(* IEC 61131-3 sources: Caravan/Stations/MachineControl/MachineControl/Class/TempControl_Class, 2 files *)

(* ---- TempControl_Class-TAB-EPM-01.st ---- *)
(*!
<Class
	Name               = "TempControl_Class"
	Revision           = "0.0"
	RealtimeTask       = "false"
	CyclicTask         = "true"
	BackgroundTask     = "false"
	Sigmatek           = "false"
	OSInterface        = "false"
	HighPriority       = "false"
	Automatic          = "false"
	UpdateMode         = "Prescan"
	SharedCommandTable = "true"
	Objectsize         = "(960,300)">
	<Channels>
		<Server Name="Actual_TempHZS_S" Visualized="true" Initialize="false" WriteProtected="false" Retentive="false"/>
		<Server Name="Actual_UltraheatTemp_S" Visualized="true" Initialize="false" WriteProtected="false" Retentive="false"/>
		<Server Name="ActualRoomTemp_S" Visualized="true" Initialize="false" WriteProtected="false" Retentive="false"/>
		<Server Name="ClassSvr" Visualized="false" Initialize="false" WriteProtected="true" Retentive="false"/>
		<Server Name="FanSpeed_S" Visualized="true" Initialize="true" DefValue="5" WriteProtected="false" Retentive="File"/>
		<Server Name="HeaterOn_S" Visualized="true" Initialize="false" WriteProtected="false" Retentive="File"/>
		<Server Name="SetRoomTemp_S" Visualized="true" Initialize="false" WriteProtected="false" Retentive="File"/>
		<Server Name="SetTempHZS_s" Visualized="true" Initialize="true" DefValue="200" WriteProtected="false" Retentive="File"/>
		<Client Name="ActualRoomTemp_C" Required="true" Internal="false"/>
		<Client Name="ActualUltraheatTemp_C" Required="true" Internal="false"/>
		<Client Name="HeaterRun_C" Required="true" Internal="false"/>
		<Client Name="MotorRunStop_C" Required="true" Internal="false"/>
		<Client Name="SetFanSpeed_C" Required="true" Internal="false"/>
		<Client Name="TempHZS_C" Required="true" Internal="false"/>
	</Channels>
</Class>
*)
TempControl_Class : CLASS
  //Servers:
	ClassSvr 	: SvrChCmd_DINT;
	Actual_TempHZS_S 	: SvrCh_DINT;
	ActualRoomTemp_S 	: SvrCh_DINT;
	Actual_UltraheatTemp_S 	: SvrCh_DINT;
	SetTempHZS_s 	: SvrCh_DINT;
	FanSpeed_S 	: SvrCh_DINT;
	SetRoomTemp_S 	: SvrCh_DINT;
	HeaterOn_S 	: SvrCh_DINT;
  //Clients:
	TempHZS_C 	: CltCh_DINT;
	ActualRoomTemp_C 	: CltCh_DINT;
	ActualUltraheatTemp_C 	: CltCh_DINT;
	SetFanSpeed_C 	: CltCh_DINT;
	MotorRunStop_C 	: CltCh_DINT;
	HeaterRun_C 	: CltCh_DINT;
  //Variables:
  //Functions:

	FUNCTION VIRTUAL GLOBAL CyWork
		VAR_INPUT
			EAX 	: UDINT;
		END_VAR
		VAR_OUTPUT
			state (EAX) 	: UDINT;
		END_VAR;
  //Tables:
	FUNCTION @STD
		VAR_OUTPUT
			ret_code	: CONFSTATES;
		END_VAR;
	FUNCTION GLOBAL TAB @CT_;
END_CLASS;

FUNCTION VIRTUAL GLOBAL TempControl_Class::CyWork
	VAR_INPUT
		EAX 	: UDINT;
	END_VAR
	VAR_OUTPUT
		state (EAX) 	: UDINT;
	END_VAR

    //Variablen einlesen
    TempHZS_C   :=    TempHZS_C.Read();

    ActualRoomTemp_C  :=  ActualRoomTemp_C.Read();

    ActualUltraheatTemp_C :=  ActualUltraheatTemp_C.Read();

    SetFanSpeed_C :=  SetFanSpeed_C.Read();

    MotorRunStop_C  :=  MotorRunStop_C.Read();

    HeaterRun_C :=  HeaterRun_C.Read();

    //Temperatur steuern
    if ActualRoomTemp_C < (SetRoomTemp_S - 1) & HeaterOn_S  = 1 then

        HeaterRun_C :=  1;

      elsif ActualRoomTemp_C > SetRoomTemp_S | HeaterOn_S = 0 then

        HeaterRun_C :=  0;

    end_if;

     //Variablen Schreiben
     Actual_TempHZS_S   :=    Actual_TempHZS_S.Write(input:=TempHZS_C);
     ActualRoomTemp_S   :=    ActualRoomTemp_S.Write(input:=ActualRoomTemp_C);

	state := READY;

END_FUNCTION

(* ---- TempControl_Class.st ---- *)
(*!
<Class
	Name               = "TempControl_Class"
	Revision           = "0.0"
	RealtimeTask       = "false"
	CyclicTask         = "true"
	BackgroundTask     = "false"
	Sigmatek           = "false"
	OSInterface        = "false"
	HighPriority       = "false"
	Automatic          = "false"
	UpdateMode         = "Prescan"
	SharedCommandTable = "true"
	Objectsize         = "(960,300)">
	<Channels>
		<Server Name="Actual_TempHZS_S" Visualized="true" Initialize="false" WriteProtected="false" Retentive="false"/>
		<Server Name="Actual_UltraheatTemp_S" Visualized="true" Initialize="false" WriteProtected="false" Retentive="false"/>
		<Server Name="ActualRoomTemp_S" Visualized="true" Initialize="false" WriteProtected="false" Retentive="false"/>
		<Server Name="ClassSvr" Visualized="false" Initialize="false" WriteProtected="true" Retentive="false"/>
		<Server Name="FanMode_S" Visualized="true" Initialize="false" WriteProtected="false" Retentive="File"/>
		<Server Name="FanSpeed_S" Visualized="true" Initialize="true" DefValue="5" WriteProtected="false" Retentive="File"/>
		<Server Name="HeaterOn_S" Visualized="true" Initialize="false" WriteProtected="false" Retentive="File"/>
		<Server Name="SetRoomTemp_S" Visualized="true" Initialize="false" WriteProtected="false" Retentive="File"/>
		<Server Name="SetTempHZS_s" Visualized="true" Initialize="true" DefValue="200" WriteProtected="false" Retentive="File"/>
		<Client Name="ActualRoomTemp_C" Required="true" Internal="false"/>
		<Client Name="ActualUltraheatTemp_C" Required="true" Internal="false"/>
		<Client Name="Heater200Watt_C" Required="true" Internal="false"/>
		<Client Name="HeaterOn_C" Required="true" Internal="false" DefValue="0"/>
		<Client Name="HeaterRun_C" Required="true" Internal="false" DefValue="0"/>
		<Client Name="MotorRunStop_C" Required="true" Internal="false"/>
		<Client Name="SetFanSpeed_C" Required="true" Internal="false"/>
		<Client Name="TempHZS_C" Required="true" Internal="false"/>
	</Channels>
</Class>
*)
TempControl_Class : CLASS
  //Servers:
	ClassSvr 	: SvrChCmd_DINT;
	Actual_TempHZS_S 	: SvrCh_DINT;
	ActualRoomTemp_S 	: SvrCh_DINT;
	Actual_UltraheatTemp_S 	: SvrCh_DINT;
	SetTempHZS_s 	: SvrCh_DINT;
	SetRoomTemp_S 	: SvrCh_DINT;
	HeaterOn_S 	: SvrCh_DINT;
	FanMode_S 	: SvrCh_DINT;
	FanSpeed_S 	: SvrCh_DINT;
  //Clients:
	TempHZS_C 	: CltCh_DINT;
	ActualRoomTemp_C 	: CltCh_DINT;
	ActualUltraheatTemp_C 	: CltCh_DINT;
	SetFanSpeed_C 	: CltCh_DINT;
	MotorRunStop_C 	: CltCh_DINT;
	HeaterRun_C 	: CltCh_DINT;
	HeaterOn_C 	: CltCh_DINT;
	Heater200Watt_C 	: CltCh_DINT;
  //Variables:
		NeedHeatRoom_VAR 	: DINT;
		NeedHeatHZS_VAR 	: DINT;
		UltraheatFanTemp_VAR 	: DINT;
		MotorSpeedCalculated_VAR 	: DINT;
  //Functions:

	FUNCTION VIRTUAL GLOBAL CyWork
		VAR_INPUT
			EAX 	: UDINT;
		END_VAR
		VAR_OUTPUT
			state (EAX) 	: UDINT;
		END_VAR;
  //Tables:
	FUNCTION @STD
		VAR_OUTPUT
			ret_code	: CONFSTATES;
		END_VAR;
	FUNCTION GLOBAL TAB @CT_;
END_CLASS;

FUNCTION VIRTUAL GLOBAL TempControl_Class::CyWork
	VAR_INPUT
		EAX 	: UDINT;
	END_VAR
	VAR_OUTPUT
		state (EAX) 	: UDINT;
	END_VAR

    //Variablen einlesen
    TempHZS_C   :=    TempHZS_C.Read();

    ActualRoomTemp_C  :=  ActualRoomTemp_C.Read();

    ActualUltraheatTemp_C :=  ActualUltraheatTemp_C.Read();

    SetFanSpeed_C :=  SetFanSpeed_C.Read();

    MotorRunStop_C  :=  MotorRunStop_C.Read();

    HeaterRun_C :=  HeaterRun_C.Read();

    //Heizung Einschalten
    if HeaterOn_S > 0 then

      HeaterOn_C  :=  HeaterOn_C.Write(input:=1);

        else

          HeaterOn_C  :=  HeaterOn_C.Write(input:=0);

    end_if;

    //Heizleistung einstellen
    if HeaterOn_S = 2 then

         Heater200Watt_C  :=  Heater200Watt_C.Write(input:=1);

       else

         Heater200Watt_C  :=  Heater200Watt_C.Write(input:=0);

    end_if;

    //Temperatur steuern Raum
    if ActualRoomTemp_C < (SetRoomTemp_S - 1) & HeaterOn_S  >= 1 then

        NeedHeatRoom_VAR :=  1;

      elsif ActualRoomTemp_C > SetRoomTemp_S | HeaterOn_S = 0 then

        NeedHeatRoom_VAR :=  0;

    end_if;

    //Temperatur steuern Schlafzimmer
    if (TempHZS_C < (SetTempHZS_s - 1)) & (HeaterOn_S  >= 1) then

        NeedHeatHZS_VAR :=  1;

      elsif TempHZS_C  >  SetTempHZS_s | HeaterOn_S = 0 then

        NeedHeatHZS_VAR :=  0;

    end_if;

    //heizung ansteuern
    if NeedHeatHZS_VAR  = 1 | NeedHeatRoom_VAR = 1 then

          HeaterRun_C :=  HeaterRun_C.Write(input:=1);

        else

          HeaterRun_C :=  HeaterRun_C.Write(input:=0);

    end_if;

    //Ventilator auf Manuell
    if FanMode_S  = 1 then

        SetFanSpeed_C   :=  SetFanSpeed_C.Write(input:=(10000/8*FanSpeed_S));

        MotorRunStop_C  :=  MotorRunStop_C.Write(input:=1);

    end_if;

    //Ventilator auf Auto

      if FanMode_S  = 2 then

          UltraheatFanTemp_VAR    :=    (ActualUltraheatTemp_C - ActualRoomTemp_C);

          MotorSpeedCalculated_VAR  :=  (10000/500*UltraheatFanTemp_VAR);

            if MotorSpeedCalculated_VAR > (10000/8*FanSpeed_S) then

                SetFanSpeed_C   :=  SetFanSpeed_C.Write(input:=(10000/8*FanSpeed_S));

              elsif MotorSpeedCalculated_VAR  >=  0 then

                SetFanSpeed_C   :=   SetFanSpeed_C.Write(input:=MotorSpeedCalculated_VAR);

              else

                SetFanSpeed_C   :=   SetFanSpeed_C.Write(input:=0);

            end_if;

        MotorRunStop_C  :=  MotorRunStop_C.Write(input:=1);

     end_if;

    //Ventilator ausschalten
    if FanMode_S  = 0 then

        MotorRunStop_C    :=    MotorRunStop_C.Write(input:=0);

    end_if;

     //Variablen Schreiben
     Actual_TempHZS_S   :=    Actual_TempHZS_S.Write(input:=TempHZS_C);
     ActualRoomTemp_S   :=    ActualRoomTemp_S.Write(input:=ActualRoomTemp_C);

	state := READY;

END_FUNCTION
